// TIA Portal V17 export
// export: Created 2026-04-13T11:12:43.3475723Z, ExportSetting WithDefaults, DisplayName Totally Integrated Automation Portal, DisplayVersion V17 Update 4, DisplayName TIA Portal Openness, DisplayVersion V17 Update 4, DisplayName TIA Portal Version Control Interface, DisplayVersion V17, DisplayName SINAMICS Startdrive Advanced, DisplayVersion V17, DisplayName SINAMICS Startdrive G130, G150, S120, S150, SINAMICS MV, S210, DisplayVersion V17, DisplayName SINAMICS Startdrive G110M, G120, G120C, G120D, G120P, G115D, DisplayVersion V17, DisplayName STEP 7 Professional, DisplayVersion V17 Update 4, DisplayName STEP 7 Safety, DisplayVersion V17, DisplayName WinCC Professional, DisplayVersion V17 Update 4
FUNCTION "LBitToWord" : Void   // FC232, SCL
TITLE = LBitToWord
{ S7_Optimized_Access := 'FALSE' }
AUTHOR : William
FAMILY : Control
VERSION : 0.1
// //============================================================================================
// //2017-04-21 15h49
// //Moves the 16 input bits to one output integer.
// //============================================================================================
// stored: AutoNumber false, IsIECCheckEnabled false, SetENOAutomatically false, UDAEnableTagReadback false
   VAR_INPUT
      I_Input0 : Bool;
      I_Input1 : Bool;
      I_Input2 : Bool;
      I_Input3 : Bool;
      I_Input4 : Bool;
      I_Input5 : Bool;
      I_Input6 : Bool;
      I_Input7 : Bool;
      I_Input8 : Bool;
      I_Input9 : Bool;
      I_Input10 : Bool;
      I_Input11 : Bool;
      I_Input12 : Bool;
      I_Input13 : Bool;
      I_Input14 : Bool;
      I_Input15 : Bool;
   END_VAR
   VAR_OUTPUT
      O_WordOut : Word;   // Output Word format
   END_VAR
   VAR_TEMP
      TempInputBit : Array[0..15] of Bool;
      TempWord AT TempInputBit : Word;
   END_VAR
BEGIN
   //============================================================================================
   //2017-04-21 15h49
   //Moves the 16 input bits to one output integer.
   //============================================================================================

   //**** 1 - Inputs ****  Move Bit to temporary bit.
   #TempInputBit[8] := #I_Input0;
   #TempInputBit[9] := #I_Input1;
   #TempInputBit[10] := #I_Input2;
   #TempInputBit[11] := #I_Input3;
   #TempInputBit[12] := #I_Input4;
   #TempInputBit[13] := #I_Input5;
   #TempInputBit[14] := #I_Input6;
   #TempInputBit[15] := #I_Input7;

   #TempInputBit[0] := #I_Input8;
   #TempInputBit[1] := #I_Input9;
   #TempInputBit[2] := #I_Input10;
   #TempInputBit[3] := #I_Input11;
   #TempInputBit[4] := #I_Input12;
   #TempInputBit[5] := #I_Input13;
   #TempInputBit[6] := #I_Input14;
   #TempInputBit[7] := #I_Input15;


   //**** 8 - Outputs **** Move the temporary Word to the output Word
   #O_WordOut := #TempWord;
END_FUNCTION
